FUNCTION_BLOCK "fbArchiveSlotTank"
{ S7_Optimized_Access := 'TRUE' }
VERSION : 0.8
   VAR
      SlotTank : Array[1..17] of Struct
         slot : Array[1..1] of "tSlot";
      END_STRUCT;
   END_VAR


BEGIN
END_FUNCTION_BLOCK

